RoboDK station: UR5_ROB2.rdk

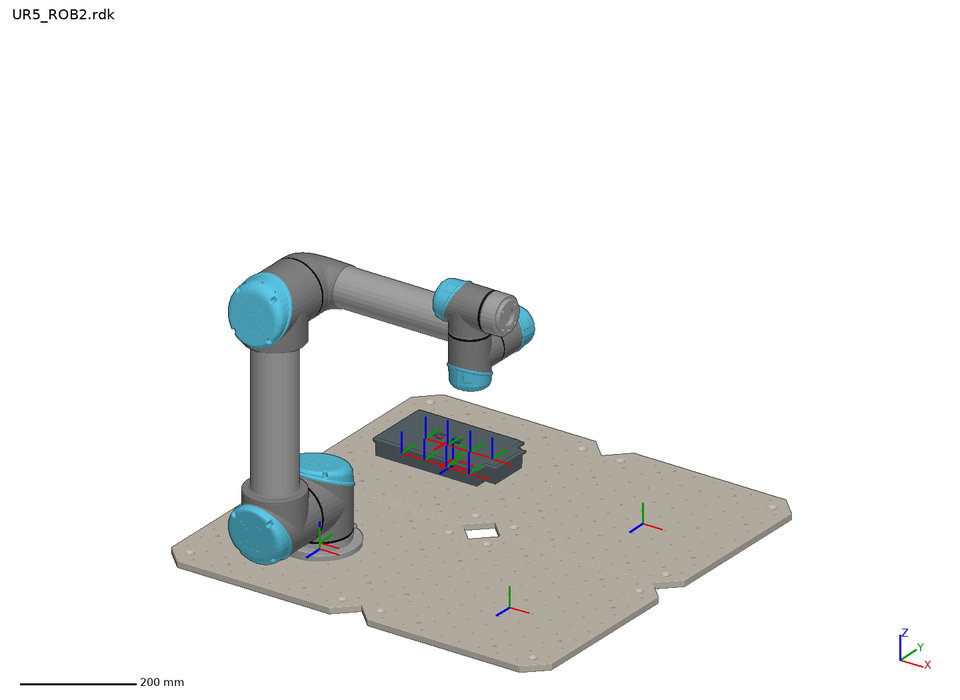
[picture v0: the station drawn from its stored meshes, robots at their saved joint values, targets as dots, program paths as lines]
Station UR5_ROB2 (saved by RoboDK 5.9.6). Poses are relative to the parent item; angles as X-Y-Z fixed-axis rotations.
  - frame UR5 Base at (0, 0, 0) mm
    - robot UR5: 6 axes
        modified DH rows (alpha deg, a mm, theta deg, d mm): 0, 0, 0, 89.2; 90, 0, 180, 0; 0, 425, 0, 0; 0, 392, 0, 109.3; -90, 0, 0, 94.75; 90, 0, 180, 82.5
        joint limits [-360, -360, -360, -360, -360, -360] to [360, 360, 360, 360, 360, 360]; home [0, -90, -90, 0, 90, 0]; saved at [0, -90, -90, 0, 90, 0]
  - frame Frame 1 at (0, 0, -12) mm, rotated rx 90 ry 0 rz 0 deg
    - object plate0x0y at (0, 0, 0) mm, size 399.5 x 12 x 399.5 mm, geometry from pallette_1x1-perforated_m6-ahl-001.STEP
  - frame Frame 2 at (400, 0, -12) mm, rotated rx 90 ry 0 rz 0 deg
    - object plate1x0y at (0, 0, 0) mm, size 399.5 x 12 x 399.5 mm, geometry from pallette_1x1-perforated_m6-ahl-001.STEP
  - frame Frame 3 at (0, 400, -12) mm, rotated rx 90 ry 0 rz 0 deg
    - object plate0x1y at (0, 0, 0) mm, size 399.5 x 12 x 399.5 mm, geometry from pallette_1x1-perforated_m6-ahl-001.STEP
  - frame Frame 4 at (400, 400, -12) mm, rotated rx 90 ry 0 rz 0 deg
    - object plate1x1y at (0, 0, 0) mm, size 399.5 x 12 x 399.5 mm, geometry from pallette_1x1-perforated_m6-ahl-001.STEP
  - frame Battery at (0, 400, 0) mm, rotated rx 0 ry 0 rz -90 deg
    - frame BatteryCase at (0, 0, 0) mm
      - object 001_BMW_Battery_Chasis_STEP at (0, 0, 0) mm, size 140 x 244 x 34 mm, geometry from 001_BMW_Battery_Chasis_STEP.stp
    - frame caseLid at (0, -10.5, 31) mm
      - object 002_BMW_Battery_Lid_ STEP at (0, 0, 0) mm, size 140 x 244 x 7 mm, geometry from 002_BMW_Battery_Lid_ STEP.stp
    - frame Cells at (0, 0, 0) mm, rotated rx 0 ry 0 rz 90 deg
      - frame 1cell at (58.5, -35.5, 3) mm
        - object 003_BMW_Module_015_F3 at (0, 0, 0) mm, size 42 x 48 x 26 mm, geometry from 003_BMW_Module_015_F3.stl
      - frame 2cell at (11.5, -35.5, 3) mm
        - object 003_BMW_Module_015_F3 at (0, 0, 0) mm, size 42 x 48 x 26 mm, geometry from 003_BMW_Module_015_F3.stl
      - frame 3cell at (-35.5, -35.5, 3) mm
        - object 003_BMW_Module_015_F3 at (0, 0, 0) mm, size 42 x 48 x 26 mm, geometry from 003_BMW_Module_015_F3.stl
      - frame 4cell at (-82.5, -35.5, 3) mm
        - object 003_BMW_Module_015_F3 at (0, 0, 0) mm, size 42 x 48 x 26 mm, geometry from 003_BMW_Module_015_F3.stl
      - frame 5cell at (58.5, 35.5, 3) mm
        - object 003_BMW_Module_015_F3 at (0, 0, 0) mm, size 42 x 48 x 26 mm, geometry from 003_BMW_Module_015_F3.stl
      - frame 6cell at (11.5, 35.5, 3) mm
        - object 003_BMW_Module_015_F3 at (0, 0, 0) mm, size 42 x 48 x 26 mm, geometry from 003_BMW_Module_015_F3.stl
      - frame 7cell at (-35.5, 35.5, 3) mm
        - object 003_BMW_Module_015_F3 at (0, 0, 0) mm, size 42 x 48 x 26 mm, geometry from 003_BMW_Module_015_F3.stl
      - frame 8cell at (-82.5, 35.5, 3) mm
        - object 003_BMW_Module_015_F3 at (0, 0, 0) mm, size 42 x 48 x 26 mm, geometry from 003_BMW_Module_015_F3.stl
